// TIA Portal V20 export
// export: Created 2025-12-01T14:56:21.6871972Z, ExportSetting None, DisplayName Totally Integrated Automation Portal, DisplayVersion V20 Update 3, DisplayName TIA Portal Openness, DisplayVersion V20 Update 3, DisplayName TIA Portal Version Control Interface, DisplayVersion V20 Update 3, DisplayName STEP 7 Professional, DisplayVersion V20 Update 3, DisplayName STEP 7 Safety, DisplayVersion V20 Update 2, DisplayName WinCC Basic/Comfort/Advanced, DisplayVersion V20 Update 3, DisplayName WinCC Professional, DisplayVersion V20 Update 3, DisplayName WinCC Unified, DisplayVersion V20 Update 3
TYPE "EstadoMaquina_MesaRodillos_DesPaletizadorCajasPlastico"
   STRUCT
      Etapa_Reset : Bool;   // Etapa MAQUINA en RESET
      Etapa_EnReposo : Bool;   // Etapa MAQUINA en REPOSO
      Etapa_EnMovimiento : Bool;   // Etapa MAQUINA en MOVIMIENTO
      Etapa_libre_03 : Bool;   // ...
      Etapa_libre_04 : Bool;   // ...
      Etapa_libre_05 : Bool;   // ...
      Etapa_libre_06 : Bool;   // ...
      Etapa_libre_07 : Bool;   // ...
      Etapa_libre_08 : Bool;   // ...
      Etapa_libre_09 : Bool;   // ...
      Etapa_libre_10 : Bool;   // ...
      Etapa_libre_11 : Bool;   // ...
      Etapa_libre_12 : Bool;   // ...
      Etapa_libre_13 : Bool;   // ...
      Etapa_libre_14 : Bool;   // ...
      Manual : Bool;   // MAQUINA EN MANUAL
      Err_Termico_MElev : Bool;   // 01. ERROR
      Err_TimeOut_SubidaMElev : Bool;   // 02. ERROR
      Err_TimeOut_BajadaMElev : Bool;   // 03. ERROR
      Err_PosicionPalas_EnReset : Bool;   // 04. ERROR
      Byte2_bit4 : Bool;   // 05. ERROR
      Byte2_bit5 : Bool;   // 06. ERROR
      Err_TimeOut_AbriendoPalaMovil : Bool;   // 07. ERROR
      Err_TimeOut_CerrandoPalaMovil : Bool;   // 08. ERROR
      Err_TimeOut_AbriendoPalaFija : Bool;   // 09. ERROR
      Err_TimeOut_CerrandoPalaFija : Bool;   // 10. ERROR
      Byte3_bit2 : Bool;   // 11. ERROR
      Byte3_bit3 : Bool;   // 12. ERROR
      Byte3_bit4 : Bool;   // 13. ERROR
      Byte3_bit5 : Bool;   // 14. ERROR
      Byte3_bit6 : Bool;   // 15. ERROR
      Byte3_bit7 : Bool;   // 16. ERROR
      Err_SegDescenso_EL : Bool;   // 17. ERROR
      Byte4_bit1 : Bool;   // 18. ERROR
      Byte4_bit2 : Bool;   // 19. ERROR
      Byte4_bit3 : Bool;   // 20. ERROR
      Byte4_bit4 : Bool;   // 21. ERROR
      Byte4_bit5 : Bool;   // 22. ERROR
      Byte4_bit6 : Bool;   // 23. ERROR
      Byte4_bit7 : Bool;   // 24. ERROR
      Byte5_bit0 : Bool;   // 25. ERROR
      Byte5_bit1 : Bool;   // 26. ERROR
      Byte5_bit2 : Bool;   // 27. ERROR
      Byte5_bit3 : Bool;   // 28. ERROR
      Byte5_bit4 : Bool;   // 29. ERROR
      Byte5_bit5 : Bool;   // 30. ERROR
      Byte5_bit6 : Bool;   // 31. ERROR
      Byte5_bit7 : Bool;   // 32. ERROR
      Byte6_bit0 : Bool;   // 33. ERROR
      Byte6_bit1 : Bool;   // 34. ERROR
      Byte6_bit2 : Bool;   // 35. ERROR
      Byte6_bit3 : Bool;   // 36. ERROR
      Byte6_bit4 : Bool;   // 37. ERROR
      Byte6_bit5 : Bool;   // 38. ERROR
      Byte6_bit6 : Bool;   // 39. ERROR
      Error_MAQx : Bool;   // Marca General Errol
      MElev_Termico : Bool;   // Entrada 1
      Byte7_bit1 : Bool;   // Entrada 2
      Byte7_bit2 : Bool;   // Entrada 3
      Byte7_bit3 : Bool;   // Entrada 4
      Byte7_bit4 : Bool;   // Entrada 5
      Byte7_bit5 : Bool;   // Entrada 6
      Byte7_bit6 : Bool;   // Entrada 7
      Byte7_bit7 : Bool;   // Entrada 8
      PosMElev_Abajo : Bool;   // Entrada 9
      PosMElev_Remotada : Bool;   // Entrada 10
      PosMElev_Paleta : Bool;   // Entrada 11
      Byte8_bit3 : Bool;   // Entrada 12
      PaletaMovil_IN : Bool;   // Entrada 13
      PaletaMovil_OUT : Bool;   // Entrada 14
      PaletaFija_IN : Bool;   // Entrada 15
      PaletaFija_OUT : Bool;   // Entrada 16
      Byte9_bit0 : Bool;   // Entrada 17
      Byte9_bit1 : Bool;   // Entrada 18
      MElev_Bamper : Bool;   // Entrada 19
      Byte9_bit3 : Bool;   // Entrada 20
      Byte9_bit4 : Bool;   // Entrada 21
      Byte9_bit5 : Bool;   // Entrada 22
      Byte9_bit6 : Bool;   // Entrada 23
      Byte9_bit7 : Bool;   // Entrada 24
      MElev_Subiendo : Bool;   // Salida 1
      MElev_Bajando : Bool;   // Salida 2
      PalaMovil_Abriendo : Bool;   // Salida 3
      PalaMovil_Cerrando : Bool;   // Salida 4
      PalaFija_Abriendo : Bool;   // Salida 5
      PalaFija_Cerrando : Bool;   // Salida 6
      Byte10_bit6 : Bool;   // Salida 7
      Byte10_bit7 : Bool;   // Salida 8
      Byte11_bit0 : Bool;   // Salida 9
      Byte11_bit1 : Bool;   // Salida 10
      Byte11_bit2 : Bool;   // Salida 11
      Byte11_bit3 : Bool;   // Salida 12
      Byte11_bit4 : Bool;   // Salida 13
      Byte11_bit5 : Bool;   // Salida 14
      Byte11_bit6 : Bool;   // Salida 15
      Byte11_bit7 : Bool;   // Salida 16
      Byte12_bit0 : Bool;   // Salida 17
      Byte12_bit1 : Bool;   // Salida 18
      Fin_VI : Bool;   // Fin de Vehiculo
      Paro_Blando : Bool;   // Maquina en paro blando
      Byte12_bit4 : Bool;   // ...
      Byte12_bit5 : Bool;   // ...
      Byte12_bit6 : Bool;   // ...
      Byte12_bit7 : Bool;   // ...
      Byte13_bit0 : Bool;   // ...
      Byte13_bit1 : Bool;   // ...
      Byte13_bit2 : Bool;   // ...
      Byte13_bit3 : Bool;   // ...
      Byte13_bit4 : Bool;   // ...
      Byte13_bit5 : Bool;   // ...
      Byte13_bit6 : Bool;   // ...
      Byte13_bit7 : Bool;   // ...
      Byte14_bit0 : Bool;   // ...
      Byte14_bit1 : Bool;   // ...
      Byte14_bit2 : Bool;   // ...
      Byte14_bit3 : Bool;   // ...
      Byte14_bit4 : Bool;   // ...
      Byte14_bit5 : Bool;   // ...
      Byte14_bit6 : Bool;   // ...
      Byte14_bit7 : Bool;   // ...
      Byte15_bit0 : Bool;   // ...
      Byte15_bit1 : Bool;   // ...
      Byte15_bit2 : Bool;   // ...
      Byte15_bit3 : Bool;   // ...
      Byte15_bit4 : Bool;   // ...
      Byte15_bit5 : Bool;   // ...
      Byte15_bit6 : Bool;   // ...
      Byte15_bit7 : Bool;   // ...
   END_STRUCT;
END_TYPE
